// TIA Portal V20 export
VAR_GLOBAL   // PLC tag table "Analog_Outputs"
   AQ_NozzleOverpressureSetPoint AT %QW428 : Word;
   AQ_FreeQW482 AT %QW430 : Word;
   AQ_VentilatorSetPoint AT %QW432 : Word;
   AQ_PropValveClimSetPoint AT %QW434 : Word;
END_VAR
